{attribute 'qualified_only'}
{attribute 'strict'}
{attribute 'to_string'}
TYPE
ApproachScenario_e :
(
    WaitOnFinishedProcess,
    WaitOnFreeStation,
    DoNotWait,
    WaitOnPrevProcess,
    WaitOnExternalTrigger,
    _MAX
);
END_TYPE

(* stored: Version 1.1.0.1, ProductVersion 3.1.4024.12
   EnumerationTextList ApproachScenario_e: Id {74f64b3a-b777-4289-aa40-9557889d62ae} *)
